ABB RobotStudio station: Solution1_20191111-121259.rsstn

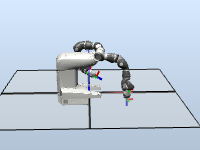
Station Solution1 (saved by RobotStudio 6.6.7701.1025)
Controller YuMi_Simfor_ROS
  mechanical unit ROB_R: IRB14000_0.5_0.5_R, 6 joints, base frame (0, 0, 0) mm
  mechanical unit ROB_R_7: IRB14000_0.5_0.5_R, 1 joints, base frame (0, 0, 0) mm
  mechanical unit ROB_L: IRB14000_0.5_0.5_L, 6 joints, base frame (0, 0, 0) mm
  mechanical unit ROB_L_7: IRB14000_0.5_0.5_L, 1 joints, base frame (0, 0, 0) mm
Layout (positions relative to the parent item):
  - IRB14000_0.5_0.5 [mechanism, from Robots\IRB14000_0.5_0.5__01.rslib] at (0, 0, 0) mm
  - IRB14000_0.5_0.5_R [mechanism, from Robots\IRB14000_0.5_0.5__01.rslib] at (0, 0, 0) mm; joint values [-0.5284, 0.6727, -0.4964, -0.2335, 4.1945, -0.1705, -1.4414] (rad or m)
  - IRB14000_0.5_0.5_L [mechanism, from Robots\IRB14000_0.5_0.5__01.rslib] at (0, 0, 0) mm; joint values [-0.0001, -2.2689, 2.3562, 0.5236, 0, 0.6982, 0.0001] (rad or m)
  - Smart_Gripper_Servo_Fingers_R [mechanism, from Tools\ABB_Smart_Gripper_Servo_Fingers.rslib] at (413.44, -193.93, 94.48) mm, rotated rx 179.66 ry -0.12 rz 14.82 deg; joint values [0] (rad or m)
  - Smart_Gripper_Servo_Fingers_L [mechanism, from Tools\ABB_Smart_Gripper_Servo_Fingers.rslib] at (-9.56, 182.6, 198.63) mm, rotated rx -179.34 ry -63.64 rz -15.46 deg; joint values [0] (rad or m)
Attachment: Smart_Gripper_Servo_Fingers_L is attached to IRB14000_0.5_0.5_L / Link7
Attachment: Smart_Gripper_Servo_Fingers_R is attached to IRB14000_0.5_0.5_R / Link7
Targets, tools, work objects and paths stored in the station, written as RAPID:
! task T_ROB_R
MODULE ROS_motion_right
  VAR syncident ready;
  PERS tasks task_list{2}:=[["T_ROB_R"],["T_ROB_L"]];
  PROC main()
    WaitSyncTask ready,task_list\TimeOut:=20;
    init_trajectory;
    MoveAbsJ target,NORM_SPEED\T:=jointTrajectory{current_index}.duration,stop_mode,tool0;
    WaitTime 0.05;
  ENDPROC
  LOCAL PROC init_trajectory()
    clear_path;
  ENDPROC
  LOCAL PROC abort_trajectory()
    clear_path;
  ENDPROC
  LOCAL PROC clear_path()
  ENDPROC
ENDMODULE

! task T_ROB_R
MODULE CalibData
  PERS tooldata Servo:=[TRUE,[[0,0,114.2],[1,0,0,0]],[0.215,[8.7,12.3,49.2],[1,0,0,0],0.00021,0.00024,0.00009]];
ENDMODULE

! task T_ROB_L
MODULE ROS_motion_left
  VAR syncident ready;
  PERS tasks task_list{2}:=[["T_ROB_R"],["T_ROB_L"]];
  PROC main()
    WaitSyncTask ready,task_list\TimeOut:=20;
    init_trajectory;
    MoveAbsJ target,NORM_SPEED\T:=jointTrajectory{current_index}.duration,stop_mode,tool0;
    WaitTime 0.05;
  ENDPROC
  LOCAL PROC init_trajectory()
    clear_path;
  ENDPROC
  LOCAL PROC abort_trajectory()
    clear_path;
  ENDPROC
  LOCAL PROC clear_path()
  ENDPROC
ENDMODULE

! task T_ROB_L
MODULE CalibData
  PERS tooldata Servo:=[TRUE,[[0,0,114.2],[1,0,0,0]],[0.215,[8.7,12.3,49.2],[1,0,0,0],0.00021,0.00024,0.00009]];
ENDMODULE

